PROGRAM MAIN
VAR
END_VAR

END_PROGRAM

(* stored: Version 1.1.0.1
   POU MAIN: Id {e26133ab-76ec-46ab-b83b-a8d9f08a4c20} *)
